PROGRAM MAIN
VAR
END_VAR

END_PROGRAM

(* stored: Version 1.1.0.1
   POU MAIN: Id {040816f1-f230-4b7f-abf9-ea3a3ab6afb7} *)
